# EPICS substitutions: hugo/source/db/Beckhoff_9XXX/ecmcEL9227-5500.substitutions
file "ecmcEL9227-5500-chx.template"
{
    pattern {CH_ID}
            {01   }
            {02   }
}
